// TwinCAT 3 PLC project Untitled1
// ProgramVersion: 3.1.4023.0
// libraries:
//   Tc2_MC2, * (Beckhoff Automation GmbH)
//   Tc2_NC, * (Beckhoff Automation GmbH)
//   Tc2_Standard, * (Beckhoff Automation GmbH)
//   Tc2_SUPS, * (Beckhoff Automation GmbH)
//   Tc2_System, * (Beckhoff Automation GmbH)
//   Tc2_Utilities, * (Beckhoff Automation GmbH)
//   Tc3_Module, * (Beckhoff Automation GmbH)
// project tree:
//   GVLs/ GVL.TcGVL
//   / PlcTask.TcTTO
//   POUs/ Axis1_Motion.TcPOU, Axis2_Motion.TcPOU, MAIN.TcPOU
//   POUs/PersistentFunction/ FB_Dummy.TcPOU (not stored), SLOWTASK.TcPOU (not stored), UPSPersitent.TcPOU (not stored)

CONFIGURATION Untitled1
    RESOURCE PLC ON TwinCAT3
        TASK PlcTask(INTERVAL := T#10ms, PRIORITY := 20);
        PROGRAM MAIN WITH PlcTask : MAIN;
        PROGRAM Axis1_FC WITH PlcTask : Axis1_FC;
        PROGRAM INIT WITH PlcTask : INIT;
        PROGRAM Axis2_FC WITH PlcTask : Axis2_FC;
    END_RESOURCE
END_CONFIGURATION

// ---- GVLs/GVL.TcGVL

VAR_GLOBAL
	//global   
	simulation:BOOL:=TRUE;
	btn_LocalOrRemote:BOOL:=FALSE;
	E_STOP  :BOOL;(*急停NC*) 
	E_STOP_In  AT%I*:BOOL;(*急停NC*) 
	E_STOP_rem:BOOL:=TRUE;//远程急停
	initStatus: BOOL;
	
	E_STOP_led :BOOL;(*急停指示*)
	Local_led  :BOOL;(*本地模式指示*)
	Remote_led :BOOL;(*远程模式指示*)
	Error:BOOL;
	ErrorId:INT;
	ErrorDescription:STRING;

	m_restartTC: BOOL;
	E_STOP_ftring:F_TRIG;
    E_STOP_rem_ftring:F_TRIG;
	
	//axis1
	axis1:AXIS_REF;
	LVDT1_IN AT%I*:INT;(*1#LVDT*)
	foreward_limit_axis1:BOOL;
	foreward_limit_axis1_In AT%I*:BOOL;//1#电机正向限位
	foreward_limit_axis1_simu:BOOL;//1#电机正向限位
	backward_limit_axis1 AT%I*:BOOL:=TRUE;//1#电机负向限位（准直器未加，默认为TRUE）
	touchLimitSwitch_axis1:BOOL;
	Axis1_error :BOOL;(*电机1故障指示*)
	Axis1_moving:BOOL;(*1#电机运行指示*)
	LVDT1_FunctionOn:BOOL;
	LVDT1_PV  :REAL;(*1#LVDT*)
	LVDT1_Threshold :REAL;
	LVDT1_OutOfThresholdRange :BOOL:=TRUE;
	LVDT1_OnceInRangeFlag :INT;
	LVDT1_ManualReleaseAlarm :BOOL;
	Axis1_Currentvelocity:REAL;
	btn_Move_Axis1: BOOL;
	btn_JogForward_Axis1: BOOL;
	btn_JogBackward_Axis1: BOOL;
	btn_Stop_Axis1: BOOL;
	btn_Reset_Axis1: BOOL;
	btn_SetPosition_Axis1:BOOL;
	Moving_done_Axis1:BOOL;
	PositionSetValue_Axis1:REAL;
	PositionSetDone_Axis1:BOOL;
	
	//axis2
	axis2:AXIS_REF;
	LVDT2_IN AT%I*:INT;(*2#LVDT*)
	foreward_limit_axis2:BOOL;
	foreward_limit_axis2_In AT%I*:BOOL;//2#电机正向限位
	foreward_limit_axis2_simu:BOOL;//1#电机正向限位
	backward_limit_axis2 AT%I*:BOOL:=TRUE;//2#电机负向限位（准直器未加，默认为TRUE）
	touchLimitSwitch_axis2:BOOL;
	Axis2_error :BOOL;(*电机2故障指示*)	 
	Axis2_moving	:BOOL;(*2#电机运行指示*)
	LVDT2_FunctionOn:	BOOL;	
	LVDT2_PV	:REAL;(*2#LVDT*)	
	LVDT2_Threshold	:REAL;	
	LVDT2_OutOfThresholdRange	:BOOL:=TRUE;	
	LVDT2_OnceInRangeFlag	:INT;	
	LVDT2_ManualReleaseAlarm	:BOOL;
	Axis2_Currentvelocity	:REAL;
	btn_Move_Axis2: BOOL;
	btn_JogForward_Axis2: BOOL;
	btn_JogBackward_Axis2: BOOL;
	btn_Stop_Axis2: BOOL;
	btn_Reset_Axis2: BOOL;
	btn_SetPosition_Axis2:BOOL;
	Moving_done_Axis2:BOOL;
	PositionSetValue_Axis2:REAL;
	PositionSetDone_Axis2:BOOL;
	
	//axis all
	btn_Move_AxisAll:BOOL;
	RTrig_Move_AxisAll:R_Trig;
	btn_Stop_AxisAll:BOOL;
	RTrig_Stop_AxisAll:R_Trig;
	btn_JogForward_AxisAll:BOOL;
	RTrig_JogForward_AxisAll:R_Trig;
	btn_JogBackward_AxisAll:BOOL;
	RTrig_JogBackward_AxisAll:R_Trig;
	btn_Reset_AxisAll:BOOL;
	RTrig_Reset_AxisAll:R_Trig;
 
	///
	///EPICS->PLC,Command
	///
	(*BOOL类型，占一个寄存器，存储16bit *)
	//1.global
	MOD_btn_LocalOrRemote						AT%MX0.0:BOOL;//12288.0  
	MOD_btn_E_STOP								AT%MX0.1:BOOL:=TRUE;//12288.1 
	MOD_m_restartTC								AT%MX0.2:BOOL;//12288.2 
	//2.axis1
	MOD_btn_Move_Axis1                          AT%MX2.0:BOOL;//12289.0
	MOD_btn_JogForward_Axis1                    AT%MX2.1:BOOL;//12289.1
	MOD_btn_JogBackward_Axis1                   AT%MX2.2:BOOL;//12289.2
	MOD_btn_Stop_Axis1                          AT%MX2.3:BOOL;//12289.3
	MOD_btn_Reset_Axis1                         AT%MX2.4:BOOL;//12289.4
	MOD_btn_SetPosition_Axis1                   AT%MX2.5:BOOL;//12289.5
	MOD_LVDT1_FunctionOn                        AT%MX2.6:BOOL;//12289.6
	MOD_LVDT1_ManualReleaseAlarm                AT%MX2.7:BOOL;//12289.7  
	MOD_btn_backup3       		                AT%MX3.0:BOOL;//12289.8
	MOD_btn_backup4			                    AT%MX3.1:BOOL;//12289.9
	MOD_btn_backup5                  			AT%MX3.2:BOOL;//12289.10
	MOD_btn_backup6                  			AT%MX3.3:BOOL;//12289.11
	MOD_btn_backup7                				AT%MX3.4:BOOL;//12289.12
	MOD_btn_backup8                         	AT%MX3.5:BOOL;//12289.13
	MOD_btn_backup9                				AT%MX3.6:BOOL;//12289.14
	MOD_btn_backup10	                        AT%MX3.7:BOOL;//12289.15
	(*REAL类型，每个值占两个寄存器*)   
	MOB_targetPositionAxis1                     AT%MB500:REAL;//12538
	MOB_targetVelocityAxis1                     AT%MB504:REAL;//12540
	MOB_increaseJogPositionAxis1                AT%MB508:REAL;//12542
	MOB_Axis1_minPosition                       AT%MB512:REAL;//12544
	MOB_Axis1_maxPosition                       AT%MB516:REAL;//12546
	MOD_LVDT1_Threshold                         AT%MB520:REAL;//12548
	MOD_PositionSetValue_Axis1					AT%MB524:REAL;//12550
	//3.axis2
	MOD_btn_Move_Axis2                          AT%MX4.0:BOOL;//12290.0
	MOD_btn_JogForward_Axis2                    AT%MX4.1:BOOL;//12290.1
	MOD_btn_JogBackward_Axis2                   AT%MX4.2:BOOL;//12290.2
	MOD_btn_Stop_Axis2                          AT%MX4.3:BOOL;//12290.3
	MOD_btn_Reset_Axis2                         AT%MX4.4:BOOL;//12290.4
	MOD_btn_SetPosition_Axis2                   AT%MX4.5:BOOL;//12290.5
	MOD_LVDT2_FunctionOn			            AT%MX4.6:BOOL;//12290.6
	MOD_LVDT2_ManualReleaseAlarm                AT%MX4.7:BOOL;//12290.7  
	MOD_btn_backup13       		                AT%MX5.0:BOOL;//12290.8
	MOD_btn_backup14			                AT%MX5.1:BOOL;//12290.9
	MOD_btn_backup15                  			AT%MX5.2:BOOL;//12290.10
	MOD_btn_backup16                  			AT%MX5.3:BOOL;//12290.11
	MOD_btn_backup17                			AT%MX5.4:BOOL;//12290.12
	MOD_btn_backup18                         	AT%MX5.5:BOOL;//12290.13
	MOD_btn_backup19                			AT%MX5.6:BOOL;//12290.14
	MOD_btn_backup20	                        AT%MX5.7:BOOL;//12290.15
	(*REAL类型，每个值占两个寄存器*)   
	MOB_targetPositionAxis2                     AT%MB600:REAL;//12588
	MOB_targetVelocityAxis2                     AT%MB604:REAL;//12590
	MOB_increaseJogPositionAxis2                AT%MB608:REAL;//12592
	MOB_Axis2_minPosition                       AT%MB612:REAL;//12594
	MOB_Axis2_maxPosition                       AT%MB616:REAL;//12596
	MOD_LVDT2_Threshold                         AT%MB620:REAL;//12598
	MOD_PositionSetValue_Axis2					AT%MB624:REAL;//12600
	//4. aixs all
	MOD_btn_Move_AxisAll                        AT%MX6.0:BOOL;//12291.0
	MOD_btn_JogForward_AxisAll                  AT%MX6.1:BOOL;//12291.1
	MOD_btn_JogBackward_AxisAll                 AT%MX6.2:BOOL;//12291.2
	MOD_btn_Stop_AxisAll                        AT%MX6.3:BOOL;//12291.3
	MOD_btn_Reset_AxisAll                       AT%MX6.4:BOOL;//12291.3
	///
	///PLC->EPICS,Response
	///
	//1.global
	(*BOOL类型，占一个寄存器，存储16bit*)
	MOD_E_STOP_led                              AT%MX10.0:BOOL;//12293.0  
	MOD_Local_led                               AT%MX10.1:BOOL;//12293.1 
	MOD_Remote_led                              AT%MX10.2:BOOL;//12293.2 
	MOD_Error_led								AT%MX10.3:BOOL;//12293.3 
	//2.axis1
	MOD_Axis1_error                             AT%MX12.0:BOOL;//12294.0
	MOD_Axis1_moving                            AT%MX12.1:BOOL;//12294.1
	MOD_foreward_limit_axis1                   	AT%MX12.2:BOOL;//12294.2
	MOD_backward_limit_axis1                    AT%MX12.3:BOOL;//12294.3
	MOD_Moving_done_Axis1                       AT%MX12.4:BOOL;//12294.4
	MOD_PositionSetDone_Axis1	                AT%MX12.5:BOOL;//12294.5
	MOD_B_Backup2	   			                AT%MX12.6:BOOL;//12294.6	
	MOD_B_Backup3	   			                AT%MX12.7:BOOL;//12294.7 
	MOD_B_Backup4                             	AT%MX13.0:BOOL;//12294.8
	MOD_B_Backup5                            	AT%MX13.1:BOOL;//12294.9
	MOD_B_Backup6                   			AT%MX13.2:BOOL;//12294.10
	MOD_B_Backup7                    			AT%MX13.3:BOOL;//12294.11
	MOD_B_Backup8                      			AT%MX13.4:BOOL;//12294.12
	MOD_B_Backup9	   			                AT%MX13.5:BOOL;//12294.13	
	MOD_B_Backup10	   			                AT%MX13.6:BOOL;//12294.14 	
	MOD_B_Backup11	   			                AT%MX13.7:BOOL;//12294.15	
	(*REAL类型，每个值占两个寄存器*) 
	MOD_Axis1_Currentvelocity                   AT%MB700:REAL;//12638
	MOD_Axis1_CurrentPosition                   AT%MB704:REAL;//12640
 	MOD_LVDT1_PV 	                            AT%MB708:REAL;//12642
	//3.axis2
	MOD_Axis2_error                             AT%MX14.0:BOOL;//12295.0
	MOD_Axis2_moving                            AT%MX14.1:BOOL;//12295.1
	MOD_foreward_limit_axis2                   	AT%MX14.2:BOOL;//12295.2
	MOD_backward_limit_axis2                    AT%MX14.3:BOOL;//12295.3
	MOD_Moving_done_Axis2                       AT%MX14.4:BOOL;//12295.4
	MOD_PositionSetDone_Axis2	                AT%MX14.5:BOOL;//12295.5
	MOD_B_Backup13	   			                AT%MX14.6:BOOL;//12295.6 	
	MOD_B_Backup14	   			                AT%MX14.7:BOOL;//12295.7	 
	MOD_B_Backup15                            	AT%MX15.0:BOOL;//12295.8
	MOD_B_Backup16                            	AT%MX15.1:BOOL;//12295.9
	MOD_B_Backup17                   			AT%MX15.2:BOOL;//12295.10
	MOD_B_Backup18                    			AT%MX15.3:BOOL;//12295.11
	MOD_B_Backup19                      		AT%MX15.4:BOOL;//12295.12
	MOD_B_Backup20	   			                AT%MX15.5:BOOL;//12295.13
	MOD_B_Backup21	   			                AT%MX15.6:BOOL;//12295.14
	MOD_B_Backup22	   			                AT%MX15.7:BOOL;//12295.15
	// REAL类型，每个值占两个寄存器  
	// REAL类型，每个值占两个寄存器  
	MOD_Axis2_Currentvelocity                	AT%MB800:REAL;//12688
	MOD_Axis2_CurrentPosition                   AT%MB804:REAL;//12690
 	MOD_LVDT2_PV                                AT%MB808:REAL;//12692
	// REAL类型，每个值占两个寄存器  
	MOD_ErrorId				                	AT%MB812:REAL;//12694
END_VAR

VAR_GLOBAL PERSISTENT
	//Axis1
    Axis1_CurrentPosition_retain:REAL;
	Axis1_minPosition		:REAL;
	Axis1_maxPosition		:REAL;
    increaseJogPositionAxis1:REAL;
	targetVelocityAxis1: REAL;
	targetPositionAxis1: REAL;
	//axis2
	Axis2_CurrentPosition_retain:REAL;
	Axis2_minPosition		:REAL;   
	Axis2_maxPosition		:REAL;
	increaseJogPositionAxis2:REAL;
	targetVelocityAxis2: REAL;
	targetPositionAxis2: REAL;
END_VAR

// ---- POUs/MAIN.TcPOU
PROGRAM MAIN
VAR
	//
	//Gloabal
	//
	RestartTC: TC_Restart;
	//
	//init
	//
	SetPosition_delay     	  :TON;
	SetPosition2getCurrentPositiondelay     	  :TON;
	init_State: INT;
	MC_SetPosition_Axis1: MC_SetPosition;
	MC_SetPosition_Axis2: MC_SetPosition;

	m_State_AxisAll: INT;
	m_delay:TON;
	init_dalay:TON;
END_VAR

//初始化，存储位置写入当前位置灯
A_init();
IF initStatus THEN
	//Axis1运动
	Axis1_Motion();
	//Axis2运动
	Axis2_Motion();
	//All Axis运动
	AxisAll_Motion();
END_IF
//是否simulation
simu();
//数据persistent存储
UPSPersitent();
//RestartTC
A_RestartTC();
//LVDT
LVDT();
//modbus
modbus();
//
limitSwicth();

ACTION A_init:
//
//0.delay
//
//
init_dalay.PT:=T#3S;
init_dalay();
init_dalay.IN:=TRUE;
IF NOT init_dalay.Q THEN
	RETURN;
END_IF
//1.初始化：加载保存的persistent变量：位置，并写入当前位置
//
init_MC();
SetPosition_delay.PT:=T#1S;
SetPosition_delay();
CASE init_State OF 
	0:
		IF NOT Axis1_moving AND NOT  Axis2_moving THEN
			init_State:=1;
		END_IF
	1:
		IF NOT initStatus THEN
			MC_SetPosition_Axis1.Position:=Axis1_CurrentPosition_retain;
			MC_SetPosition_Axis2.Position:=	Axis2_CurrentPosition_retain;
			MC_SetPosition_Axis1.Execute:=TRUE;
			MC_SetPosition_Axis2.Execute:=TRUE;
			SetPosition_delay.IN:=TRUE;
			init_State:=2;
		END_IF
	2:
		IF MC_SetPosition_Axis1.Done AND MC_SetPosition_Axis2.Done THEN
			init_State:=88;
		END_IF
		IF SetPosition_delay.Q THEN//延时结束时，还没有设置位置成功
			init_State:=-100;
		END_IF
	88:
		initStatus:=TRUE;
		MC_SetPosition_Axis1.Execute:=FALSE;
		MC_SetPosition_Axis2.Execute:=FALSE;
		SetPosition_delay.IN:=FALSE;
		init_State:=0;
	-100:
		initStatus:=FALSE;
		SetPosition_delay.IN:=FALSE;
		MC_SetPosition_Axis1.Execute:=FALSE;
		MC_SetPosition_Axis2.Execute:=FALSE;
		Error:=TRUE;
		ErrorId:=1;
		ErrorDescription:='init fail';
END_CASE

//
//2.位置写入后，当前位置和速度即从轴中获取
//
IF initStatus THEN
	Axis1_CurrentPosition_retain  :=LREAL_TO_REAL(axis1.NcToPlc.ActPos);
	Axis1_Currentvelocity  :=LREAL_TO_REAL(axis1.NcToPlc.ActVelo);
	Axis2_CurrentPosition_retain  :=LREAL_TO_REAL(axis2.NcToPlc.ActPos);
	Axis2_Currentvelocity  :=LREAL_TO_REAL(axis2.NcToPlc.ActVelo);
END_IF
END_ACTION

ACTION A_RestartTC:
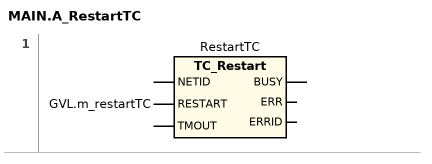
// NETWORK 1
RestartTC(RESTART := GVL.m_restartTC); // TC_Restart
END_ACTION

ACTION AxisAll_Motion:
RTrig_Move_AxisAll(CLK:=btn_Move_AxisAll,Q=>);
IF RTrig_Move_AxisAll.Q THEN
	btn_Move_Axis1:=TRUE;
	btn_Move_Axis2:=TRUE;
END_IF

RTrig_Stop_AxisAll(CLK:=btn_Stop_AxisAll,Q=>);
IF RTrig_Stop_AxisAll.Q THEN
	btn_Stop_Axis1:=TRUE;
	btn_Stop_Axis2:=TRUE;
END_IF
RTrig_JogForward_AxisAll(CLK:=btn_JogForward_AxisAll,Q=>);
IF RTrig_JogForward_AxisAll.Q THEN
	btn_JogForward_Axis1:=TRUE;
	btn_JogForward_Axis2:=TRUE;
END_IF
RTrig_JogBackward_AxisAll(CLK:=btn_JogBackward_AxisAll,Q=>);
IF RTrig_JogBackward_AxisAll.Q THEN
	btn_JogBackward_Axis1:=TRUE;
	btn_JogBackward_Axis2:=TRUE;
END_IF
RTrig_Reset_AxisAll(CLK:=btn_Reset_AxisAll,Q=>);
IF RTrig_Reset_AxisAll.Q THEN
	btn_Reset_Axis1:=TRUE;
	btn_Reset_Axis2:=TRUE;
END_IF
END_ACTION

ACTION init_MC:
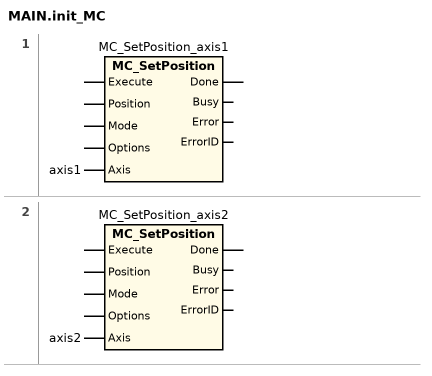
// NETWORK 1
MC_SetPosition_axis1(Axis := axis1); // MC_SetPosition

// NETWORK 2
MC_SetPosition_axis2(Axis := axis2); // MC_SetPosition
END_ACTION

ACTION limitSwicth:
touchLimitSwitch_axis1:=foreward_limit_axis1 AND backward_limit_axis1;
touchLimitSwitch_axis2:=foreward_limit_axis2 AND backward_limit_axis2;
END_ACTION

ACTION LVDT:
LVDT1_PV:=INT_TO_REAL(LVDT1_IN);
LVDT2_PV:=INT_TO_REAL(LVDT2_IN);
//LVDT1
IF LVDT1_FunctionOn THEN
	IF LVDT1_PV<=LVDT1_Threshold THEN//进入传感器限位区，报错
		LVDT1_OutOfThresholdRange:=FALSE;
		Error:=TRUE;
		ErrorDescription:='LVDT1 In Alarm Range';
		LVDT1_OnceInRangeFlag:=1;//标志曾经进入过限位区
	END_IF
	//正常情况下，出限位区，恢复正常
	//如果曾经进入过限位区，需要手动解除后，报警才解除
	IF LVDT1_OnceInRangeFlag=1 THEN
		LVDT1_OutOfThresholdRange:=FALSE;
		Error:=TRUE;
		ErrorDescription:='LVDT1 In Alarm Range';
		IF LVDT1_ManualReleaseAlarm THEN
			Error:=FALSE;
			ErrorDescription:='';
			LVDT1_OnceInRangeFlag:=0;
			LVDT1_ManualReleaseAlarm:=FALSE;
			LVDT1_OutOfThresholdRange:=TRUE;
		END_IF
	END_IF
END_IF
//LVDT2
IF LVDT2_FunctionOn THEN
	IF LVDT2_PV<=LVDT2_Threshold THEN//进入传感器限位区，报错
		LVDT2_OutOfThresholdRange:=FALSE;
		Error:=TRUE;
		ErrorDescription:='LVDT2 In Alarm Range';
		LVDT2_OnceInRangeFlag:=1;//标志曾经进入过限位区
	END_IF
	//正常情况下，出限位区，恢复正常
	//如果曾经进入过限位区，需要手动解除后，报警才解除
	IF LVDT2_OnceInRangeFlag=1 THEN
		LVDT2_OutOfThresholdRange:=FALSE;
		Error:=TRUE;
		ErrorDescription:='LVDT2 In Alarm Range';
		IF LVDT2_ManualReleaseAlarm THEN
			Error:=FALSE;
			ErrorDescription:='';
			LVDT2_OnceInRangeFlag:=0;
			LVDT2_ManualReleaseAlarm:=FALSE;
			LVDT2_OutOfThresholdRange:=TRUE;
		END_IF
	END_IF
END_IF
END_ACTION

ACTION modbus:
//PLC->EPICS，持续通讯
MOD_E_STOP_led            			:=E_STOP_led;
MOD_Axis1_error            			:=Axis1_error;
MOD_Axis2_error            			:=Axis2_error;
MOD_Axis1_moving           			:=Axis1_moving;
MOD_Axis2_moving           			:=Axis2_moving;
MOD_Moving_done_Axis1      			:=Moving_done_Axis1;
MOD_Moving_done_Axis2     			:=Moving_done_Axis2;
MOD_foreward_limit_axis1   			:=foreward_limit_axis1;
MOD_backward_limit_axis1   			:=backward_limit_axis1;
MOD_foreward_limit_axis2   			:=foreward_limit_axis2;
MOD_backward_limit_axis2   			:=backward_limit_axis2;
MOD_Axis1_Currentvelocity  			:=Axis1_Currentvelocity;
MOD_Axis2_Currentvelocity  			:=Axis2_Currentvelocity;
MOD_Axis1_CurrentPosition  			:=Axis1_CurrentPosition_retain;
MOD_Axis2_CurrentPosition  			:=Axis2_CurrentPosition_retain;
MOD_LVDT1_PV               			:=LVDT1_PV;
MOD_LVDT2_PV               			:=LVDT2_PV;
MOD_PositionSetDone_Axis1			:=PositionSetDone_Axis1;
MOD_PositionSetDone_Axis2			:=PositionSetDone_Axis2;
MOD_Error_led						:=Error;
MOD_ErrorId							:=ErrorId;
//EPICS->PLC，持续通讯
//btn_LocalOrRemote					:=MOD_btn_LocalOrRemote;

//本地模式切换
IF btn_LocalOrRemote THEN
	Local_led:= TRUE;
	Remote_led:=FALSE;
ELSE	
	Local_led:= FALSE;
	Remote_led:=TRUE;
END_IF;
MOD_Local_led:=Local_led;
MOD_Remote_led:=Remote_led;
//远程开关开，通讯
IF  MOD_Remote_led  THEN   
	//global 
	m_restartTC						:=MOD_m_restartTC;
	E_STOP_rem						:=MOD_btn_E_STOP;
	//axis1
	LVDT1_FunctionOn             	:=MOD_LVDT1_FunctionOn;    
	LVDT1_ManualReleaseAlarm     	:=MOD_LVDT1_ManualReleaseAlarm; 
	btn_SetPosition_Axis1           :=MOD_btn_SetPosition_Axis1;
	targetPositionAxis1				:=MOB_targetPositionAxis1;
	targetVelocityAxis1				:=MOB_targetVelocityAxis1;
	increaseJogPositionAxis1		:=MOB_increaseJogPositionAxis1;
	Axis1_minPosition				:=MOB_Axis1_minPosition;
	Axis1_maxPosition				:=MOB_Axis1_maxPosition;
	LVDT1_Threshold             	:=MOD_LVDT1_Threshold;
	PositionSetValue_Axis1			:=MOD_PositionSetValue_Axis1;
	//axis2
	LVDT2_Threshold              	:=MOD_LVDT2_Threshold;
	LVDT2_FunctionOn             	:=MOD_LVDT2_FunctionOn;    
	LVDT2_ManualReleaseAlarm    	:=MOD_LVDT2_ManualReleaseAlarm; 
	btn_SetPosition_Axis2           :=MOD_btn_SetPosition_Axis2;
	targetPositionAxis2				:=MOB_targetPositionAxis2;
	targetVelocityAxis2				:=MOB_targetVelocityAxis2;
	increaseJogPositionAxis2		:=MOB_increaseJogPositionAxis2;
	Axis2_minPosition				:=MOB_Axis2_minPosition;
	Axis2_maxPosition				:=MOB_Axis2_maxPosition;
	LVDT2_Threshold             	:=MOD_LVDT2_Threshold;
	PositionSetValue_Axis2			:=MOD_PositionSetValue_Axis2;
	//axis all
	btn_Move_AxisAll				:=MOD_btn_Move_AxisAll;
	btn_JogForward_AxisAll			:=MOD_btn_JogForward_AxisAll;
	btn_JogBackward_AxisAll			:=MOD_btn_JogBackward_AxisAll;
	btn_Stop_AxisAll				:=MOD_btn_Stop_AxisAll;
	IF NOT MOD_btn_Move_AxisAll	THEN
			btn_Move_Axis1                	:=MOD_btn_Move_Axis1;
			btn_Move_Axis2                	:=MOD_btn_Move_Axis2;
	ELSE
		btn_Move_AxisAll:=TRUE;
	END_IF
		IF NOT MOD_btn_Stop_AxisAll	THEN
			btn_Stop_Axis1                	:=MOD_btn_Stop_Axis1;
			btn_Stop_Axis2                	:=MOD_btn_Stop_Axis2;
	ELSE
		btn_Stop_AxisAll:=TRUE;
	END_IF
	IF NOT MOD_btn_JogForward_AxisAll	THEN
			btn_JogForward_Axis1              :=MOD_btn_JogForward_Axis1;
			btn_JogForward_Axis2              :=MOD_btn_JogForward_Axis2;
	ELSE
		btn_JogForward_AxisAll:=TRUE;
	END_IF
	IF NOT MOD_btn_JogBackward_AxisAll	THEN
			btn_JogBackward_Axis1                	:=MOD_btn_JogBackward_Axis1;
			btn_JogBackward_Axis2                	:=MOD_btn_JogBackward_Axis2;
	ELSE
		btn_JogBackward_AxisAll:=TRUE;
	END_IF
	IF NOT MOD_btn_Reset_AxisAll	THEN
			btn_Reset_Axis1                	:=MOD_btn_Reset_Axis1;
			btn_Reset_Axis2                	:=MOD_btn_Reset_Axis2;
	ELSE
		btn_Reset_AxisAll:=TRUE;
	END_IF
ELSE
	MOB_Axis1_minPosition				:=Axis1_minPosition;
	MOB_Axis1_maxPosition				:=Axis1_maxPosition;
	MOB_Axis2_minPosition				:=Axis2_minPosition;
	MOB_Axis2_maxPosition				:=Axis2_maxPosition;
	MOB_targetPositionAxis1				:=targetPositionAxis1;
	MOB_targetVelocityAxis1				:=targetVelocityAxis1;
	MOB_increaseJogPositionAxis1		:=increaseJogPositionAxis1;
	MOB_targetPositionAxis2				:=targetPositionAxis2;
	MOB_targetVelocityAxis2				:=targetVelocityAxis2;
	MOB_increaseJogPositionAxis2		:=increaseJogPositionAxis2;
END_IF
END_ACTION

ACTION simu:
IF simulation THEN
	E_STOP:=TRUE;
	foreward_limit_axis1:=TRUE;
	foreward_limit_axis2:=TRUE;
ELSE
	E_STOP:=E_STOP_In;
	foreward_limit_axis1:=foreward_limit_axis1_In;
	foreward_limit_axis2:=foreward_limit_axis2_In;
END_IF
END_ACTION

END_PROGRAM

// ---- POUs/Axis1_Motion.TcPOU
PROGRAM Axis1_Motion
VAR
	//power
	MC_Power_Axis1: MC_Power;
	//Move
	m_State_Axis1: INT;
	MC_MoveAbsolute_Axis1: MC_MoveAbsolute;

	//JOG
	j_State_Axis1: INT;
	MC_JOG_Axis1: MC_Jog;

	//Stop
	MC_Stop_Axis1: MC_Stop;
	s_State_Axis1: INT;

	//reset
	r_State_Axis1: INT;
	MC_Reset_Axis1: MC_Reset;

	//setposition
	MC_SetPosition_Axis1: MC_SetPosition;
	sp_State_Axis1: INT;
	SetPosition_delay_Axis1:TON;

	//button interlock
	Axis1_J1: BOOL;//JOG+
	Axis1_J2: BOOL;//JOG-
	Axis1_P: BOOL;//Position moving
	Axis1_S: BOOL;//Stop
	Axis1_SP: BOOL;//set position
	//input protect
	Axis1_PositionProtectionSet:BOOL;
	Axis1_InputPositionOutOfRange:BOOL;
END_VAR

//
//输入保护
//
IF targetPositionAxis1>=Axis1_minPosition AND targetPositionAxis1<=Axis1_maxPosition THEN
	Axis1_InputPositionOutOfRange:=FALSE;
	Error:=FALSE;
	ErrorId:=0;
	ErrorDescription:='';
ELSE
	Axis1_InputPositionOutOfRange:=TRUE;
	Error:=TRUE;
	ErrorId:=1001;
	ErrorDescription:='Axis1_InputPositionOutOfRange';
	RETURN;
END_IF
//
//运行状态指示
//
Axis1.ReadStatus();
IF  Axis1.Status.Moving  THEN
	Axis1_moving:=TRUE;
ELSE
	Axis1_moving:=FALSE;
END_IF;
//
//电机错误指示
//
IF  axis1.NcToPlc.ErrorCode=0 THEN
	Axis1_error     := FALSE;
ELSE
	Axis1_error     := TRUE;
	Error:=TRUE;
	ErrorId:=1002;
	ErrorDescription:='axis1.NcToPlc.ErrorCode=0';
END_IF;
//
//Moving_done_Axis1
//
//
Moving_done_Axis1:=MC_MoveAbsolute_Axis1.Done OR MC_JOG_Axis1.Done;

//Positioning move
//
A_MCAxis1();
CASE m_State_Axis1 OF 
	0:
		//检查是否有错误等
		IF  E_STOP  AND NOT Axis1_error THEN
			m_State_Axis1:=1;
		ELSE
			m_State_Axis1:=-100;
		END_IF
	1:
		//检查电机是否已经上电，如无，则上电
		IF 	NOT MC_Power_Axis1.Status THEN
			MC_Power_Axis1.Enable:=TRUE;
		ELSE
			m_State_Axis1:=2;
		END_IF
	2:
		//定位运行
		MC_MoveAbsolute_Axis1.Position:=targetPositionAxis1;
		MC_MoveAbsolute_Axis1.Velocity:=targetVelocityAxis1;
		IF btn_Move_Axis1 THEN
			MC_MoveAbsolute_Axis1.Execute:=TRUE;
			m_State_Axis1:=3;
		END_IF
	3:
		//是否运动到位
		IF MC_MoveAbsolute_Axis1.Done THEN
			m_State_Axis1:=88;
		END_IF
	88:
		btn_Move_Axis1:=FALSE;
		MC_MoveAbsolute_Axis1.Execute:=FALSE;
		m_State_Axis1:=0;		
	-100:
		btn_Move_Axis1:=FALSE;
		MC_MoveAbsolute_Axis1.Execute:=FALSE;
		Error:=TRUE;
		ErrorId:=1002;
		ErrorDescription:='E_STOP AND NOT Axis1_error';
		
END_CASE
//
//JOG+
//
CASE j_State_Axis1 OF 
	0:
		//检查是否有错误等
		IF  E_STOP  AND NOT Axis1_error THEN
			j_State_Axis1:=1;
		ELSE
			j_State_Axis1:=-100;
		END_IF
	1:
		//检查电机是否已经上电，如无，则上电
		IF 	NOT MC_Power_Axis1.Status THEN
			MC_Power_Axis1.Enable:=TRUE;
		ELSE
			j_State_Axis1:=2;
		END_IF
	2:
		//JOG运行
		MC_JOG_Axis1.Position:=increaseJogPositionAxis1;
		MC_JOG_Axis1.Velocity:=targetVelocityAxis1;
		IF btn_JogForward_Axis1 AND NOT btn_JogBackward_Axis1 THEN
			MC_JOG_Axis1.JogForward:=TRUE;
			j_State_Axis1:=3;
		END_IF
		IF btn_JogBackward_Axis1 AND NOT btn_JogForward_Axis1 THEN
			MC_JOG_Axis1.JogBackwards:=TRUE;
			j_State_Axis1:=3;
		END_IF
	3:
		//是否运动到位
		IF btn_JogForward_Axis1 THEN
			btn_JogForward_Axis1:=FALSE;
		END_IF 
		IF btn_JogBackward_Axis1 THEN
			btn_JogBackward_Axis1:=FALSE;
		END_IF
		IF MC_JOG_Axis1.Done THEN
			j_State_Axis1:=88;
		END_IF
	88:
		MC_JOG_Axis1.JogForward:=FALSE;
		MC_JOG_Axis1.JogBackwards:=FALSE;
		btn_JogForward_Axis1:=FALSE;
		btn_JogBackward_Axis1:=FALSE;
		j_State_Axis1:=0;	
		
	-100:
		MC_JOG_Axis1.JogForward:=FALSE;
		MC_JOG_Axis1.JogBackwards:=FALSE;
		btn_JogForward_Axis1:=FALSE;
		btn_JogBackward_Axis1:=FALSE;
		Error:=TRUE;
		ErrorId:=1002;
		ErrorDescription:='E_STOP AND NOT Axis1_error';	
END_CASE
//
//STOP
//
CASE s_State_Axis1 OF 
	0:
		//检查是否有错误等
		IF  E_STOP  AND NOT Axis1_error THEN
			s_State_Axis1:=1;
		ELSE
			s_State_Axis1:=-100;
		END_IF
	1:
		//检查电机是否已经上电，如无，则上电
		IF 	NOT MC_Power_Axis1.Status THEN
			MC_Power_Axis1.Enable:=TRUE;
		ELSE
			s_State_Axis1:=2;
		END_IF
	2:
		//STOP
		IF btn_Stop_Axis1 THEN
			MC_Stop_Axis1.Execute:=TRUE;
			s_State_Axis1:=3;
		END_IF
	3:
		//是否运动到位
		IF MC_Stop_Axis1.Done THEN
			s_State_Axis1:=88;
		END_IF
	88:
		btn_Stop_Axis1:=FALSE;
		MC_Stop_Axis1.Execute:=FALSE;
		s_State_Axis1:=0;	
		//reset status
		btn_Move_Axis1:=FALSE;
		MC_MoveAbsolute_Axis1.Execute:=FALSE;
		btn_JogForward_Axis1:=FALSE;
		btn_JogBackward_Axis1:=FALSE;
		MC_JOG_Axis1.JogForward:=FALSE;
		MC_JOG_Axis1.JogBackwards:=FALSE;
		m_State_Axis1:=0;
		j_State_Axis1:=0;
	-100:
		btn_Stop_Axis1:=FALSE;
		MC_Stop_Axis1.Execute:=FALSE;
		Error:=TRUE;
		ErrorId:=1002;
		ErrorDescription:='E_STOP AND NOT Axis1_error';
		//reset status
		btn_Move_Axis1:=FALSE;
		MC_MoveAbsolute_Axis1.Execute:=FALSE;
		btn_JogForward_Axis1:=FALSE;
		btn_JogBackward_Axis1:=FALSE;
		MC_JOG_Axis1.JogForward:=FALSE;
		MC_JOG_Axis1.JogBackwards:=FALSE;
		m_State_Axis1:=0;
		j_State_Axis1:=0;
END_CASE
//
//Reset
//
CASE r_State_Axis1 OF 
	0:
		IF btn_Reset_Axis1 THEN
			MC_Reset_Axis1.Execute:=TRUE;
			r_State_Axis1:=1;
		END_IF
	1:
		//是否运动到位
		IF MC_Reset_Axis1.Done THEN
			r_State_Axis1:=88;
		END_IF
	88:
		r_State_Axis1:=0;
		MC_Reset_Axis1.Execute:=FALSE;	
		btn_Reset_Axis1:=FALSE;
		//reset status
		btn_Move_Axis1:=FALSE;
		MC_MoveAbsolute_Axis1.Execute:=FALSE;
		btn_JogForward_Axis1:=FALSE;
		btn_JogBackward_Axis1:=FALSE;
		MC_JOG_Axis1.JogForward:=FALSE;
		MC_JOG_Axis1.JogBackwards:=FALSE;
		m_State_Axis1:=0;
		s_State_Axis1:=0;
		j_State_Axis1:=0;
END_CASE
//
//setposotion
//
SetPosition_delay_Axis1.PT:=T#0.1S;
SetPosition_delay_Axis1();
IF btn_SetPosition_Axis1 THEN
	CASE sp_State_Axis1 OF 
		0:
			IF NOT Axis1_moving THEN
				sp_State_Axis1:=1;
			END_IF
		1:
			MC_SetPosition_Axis1.Position:=PositionSetValue_Axis1;
			MC_SetPosition_Axis1.Execute:=TRUE;
			SetPosition_delay_Axis1.IN:=TRUE;
			sp_State_Axis1:=2;
		2:
			IF MC_SetPosition_Axis1.Done THEN
				sp_State_Axis1:=88;
			END_IF
			IF SetPosition_delay_Axis1.Q THEN//延时结束时，还没有设置位置成功
				sp_State_Axis1:=-100;
			END_IF
		88:
			PositionSetDone_Axis1:=TRUE;
			MC_SetPosition_Axis1.Execute:=FALSE;
			SetPosition_delay_Axis1.IN:=FALSE;
			sp_State_Axis1:=0;
			btn_SetPosition_Axis1:=FALSE;
		-100:
			PositionSetDone_Axis1:=FALSE;
			MC_SetPosition_Axis1.Execute:=FALSE;
			SetPosition_delay_Axis1.IN:=FALSE;
			btn_SetPosition_Axis1:=FALSE;
	END_CASE
END_IF
//
//屏幕按钮**互锁变量,FALSE时，该按钮灰色不能触发
//
//J1->JOG+
IF  foreward_limit_axis1 AND E_STOP  AND Local_led AND NOT  Axis1_error  AND NOT  Axis1_moving AND
	NOT btn_Move_Axis1 AND NOT  btn_JogBackward_Axis1  THEN
	Axis1_J1     := TRUE;
ELSE
	Axis1_J1     := FALSE;
END_IF;
//J2>JOG-
IF  backward_limit_axis1  AND E_STOP   AND Local_led AND NOT  Axis1_error  AND NOT  Axis1_moving AND 
	 NOT  btn_Move_Axis1 AND NOT btn_JogForward_Axis1 THEN
	Axis1_J2     := TRUE;
ELSE
	Axis1_J2     := FALSE;
END_IF;
//P->PositionMove
IF  E_STOP   AND Local_led AND NOT  Axis1_error  AND NOT  Axis1_moving AND 
	 NOT btn_JogForward_Axis1  AND NOT  btn_JogBackward_Axis1 THEN
	Axis1_P     := TRUE;
ELSE
	Axis1_P     := FALSE;
END_IF;
//SP->SetPosition
IF E_STOP  AND Local_led AND NOT  Axis1_error  AND NOT Axis1_moving  THEN
	Axis1_SP     := TRUE;
ELSE
	Axis1_SP     := FALSE;
END_IF;
//S->Stop
IF E_STOP  AND Local_led AND NOT  Axis1_error THEN
	Axis1_S     := TRUE;
ELSE
	Axis1_S     := FALSE;
END_IF;
//
//
//
//急停
E_STOP_ftring(CLK:=E_STOP , Q=> );
E_STOP_rem_ftring(CLK:=E_STOP_rem , Q=> );
IF E_STOP_ftring.Q OR E_STOP_rem_ftring.Q THEN     
	E_STOP_led:= TRUE;	
	MC_Power_Axis1.Enable:=FALSE;//电机1断电
	btn_Stop_Axis1:=TRUE;//STOP axis1
	A_MCAxis1();
	Error:=TRUE;
	ErrorId:=101;
	ErrorDescription:='E_STOP';
END_IF;

ACTION A_MCAxis1:
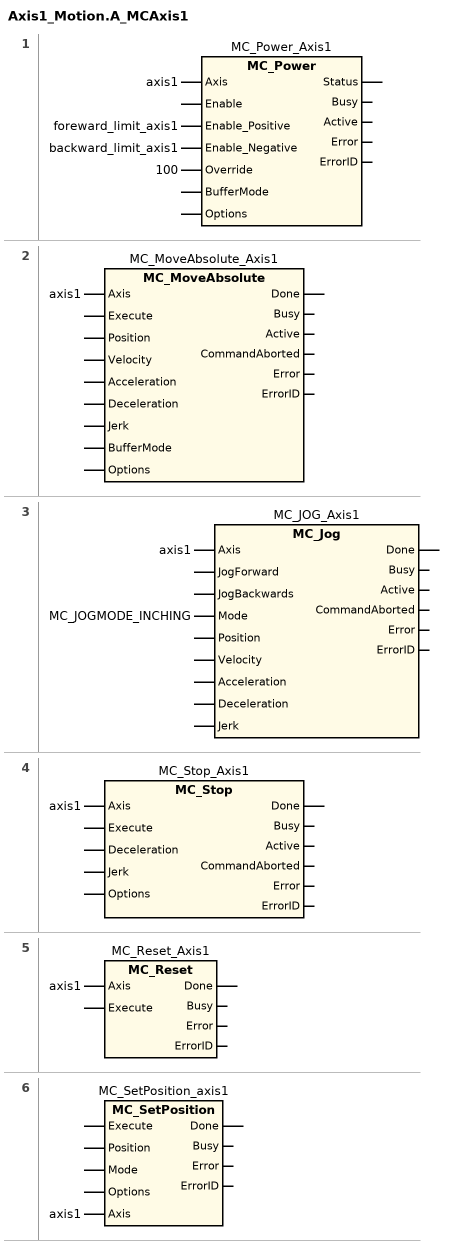
// NETWORK 1
MC_Power_Axis1(
    Axis := axis1,
    Enable_Positive := foreward_limit_axis1,
    Enable_Negative := backward_limit_axis1,
    Override := 100); // MC_Power

// NETWORK 2
MC_MoveAbsolute_Axis1(Axis := axis1); // MC_MoveAbsolute

// NETWORK 3
MC_JOG_Axis1(Axis := axis1, Mode := MC_JOGMODE_INCHING); // MC_Jog

// NETWORK 4
MC_Stop_Axis1(Axis := axis1); // MC_Stop

// NETWORK 5
MC_Reset_Axis1(Axis := axis1); // MC_Reset

// NETWORK 6
MC_SetPosition_axis1(Axis := axis1); // MC_SetPosition
END_ACTION

END_PROGRAM

// ---- POUs/Axis2_Motion.TcPOU
PROGRAM Axis2_Motion
VAR
	//power
	MC_Power_Axis2: MC_Power;
	//Move
	m_State_Axis2: INT;
	MC_MoveAbsolute_Axis2: MC_MoveAbsolute;

	//JOG
	j_State_Axis2: INT;
	MC_JOG_Axis2: MC_Jog;

	//Stop
	MC_Stop_Axis2: MC_Stop;
	s_State_Axis2: INT;

	//reset
	r_State_Axis2: INT;
	MC_Reset_Axis2: MC_Reset;

	//setposition
	MC_SetPosition_Axis2: MC_SetPosition;
	sp_State_Axis2: INT;
	SetPosition_delay_Axis2:TON;
	//button interlock
	Axis2_J1: BOOL;//JOG+
	Axis2_J2: BOOL;//JOG-
	Axis2_P: BOOL;//Position moving
	Axis2_S: BOOL;//Stop
	Axis2_SP: BOOL;//set position
	//input protect
	Axis2_PositionProtectionSet:BOOL;
	Axis2_InputPositionOutOfRange:BOOL;	
	//
END_VAR

//
//输入保护
//
IF targetPositionAxis2>=Axis2_minPosition AND targetPositionAxis2<=Axis2_maxPosition THEN
	Axis2_InputPositionOutOfRange:=FALSE;
	Error:=FALSE;
	ErrorId:=0;
	ErrorDescription:='';
ELSE
	Axis2_InputPositionOutOfRange:=TRUE;
	Error:=TRUE;
	ErrorId:=1001;
	ErrorDescription:='Axis2_InputPositionOutOfRange';
	RETURN;
END_IF
//
//运行状态指示
//
Axis2.ReadStatus();
IF  Axis2.Status.Moving  THEN
	Axis2_moving:=TRUE;
ELSE
	Axis2_moving:=FALSE;
END_IF;
//
//电机错误指示
//
IF  axis2.NcToPlc.ErrorCode=0 THEN
	Axis2_error     := FALSE;
ELSE
	Axis2_error     := TRUE;
	Error:=TRUE;
	ErrorId:=1002;
	ErrorDescription:='axis1.NcToPlc.ErrorCode=0';
END_IF;
//
//Moving_done_Axis2
//
//
Moving_done_Axis2:=MC_MoveAbsolute_Axis2.Done OR MC_JOG_Axis2.Done;
//
//Positioning move
//
A_MCAxis2();
CASE m_State_Axis2 OF 
	0:
		//检查是否有错误等
		IF  E_STOP  AND NOT Axis2_error THEN
			m_State_Axis2:=1;
		ELSE
			m_State_Axis2:=-100;
		END_IF
	1:
		//检查电机是否已经上电，如无，则上电
		IF 	NOT MC_Power_Axis2.Status THEN
			MC_Power_Axis2.Enable:=TRUE;
		ELSE
			m_State_Axis2:=2;
		END_IF
	2:
		//定位运行
		MC_MoveAbsolute_Axis2.Position:=targetPositionAxis2;
		MC_MoveAbsolute_Axis2.Velocity:=targetVelocityAxis2;
		IF btn_Move_Axis2 THEN
			MC_MoveAbsolute_Axis2.Execute:=TRUE;
			m_State_Axis2:=3;
		END_IF
	3:
		//是否运动到位
		IF MC_MoveAbsolute_Axis2.Done THEN
			m_State_Axis2:=88;
		END_IF
	88:
		btn_Move_Axis2:=FALSE;
		MC_MoveAbsolute_Axis2.Execute:=FALSE;
		m_State_Axis2:=0;		
	-100:
		btn_Move_Axis2:=FALSE;
		MC_MoveAbsolute_Axis2.Execute:=FALSE;
		Error:=TRUE;
		ErrorId:=1002;
		ErrorDescription:='E_STOP AND NOT Axis2_error';
		
END_CASE
//
//JOG+
//
CASE j_State_Axis2 OF 
	0:
		//检查是否有错误等
		IF  E_STOP  AND NOT Axis2_error THEN
			j_State_Axis2:=1;
		ELSE
			j_State_Axis2:=-100;
		END_IF
	1:
		//检查电机是否已经上电，如无，则上电
		IF 	NOT MC_Power_Axis2.Status THEN
			MC_Power_Axis2.Enable:=TRUE;
		ELSE
			j_State_Axis2:=2;
		END_IF
	2:
		//JOG运行
		MC_JOG_Axis2.Position:=increaseJogPositionAxis2;
		MC_JOG_Axis2.Velocity:=targetVelocityAxis2;
		IF btn_JogForward_Axis2 AND NOT btn_JogBackward_Axis2 THEN
			MC_JOG_Axis2.JogForward:=TRUE;
			j_State_Axis2:=3;
		END_IF
		IF btn_JogBackward_Axis2 AND NOT btn_JogForward_Axis2 THEN
			MC_JOG_Axis2.JogBackwards:=TRUE;
			j_State_Axis2:=3;
		END_IF
	3:
		//是否运动到位
		IF btn_JogForward_Axis2 THEN
			btn_JogForward_Axis2:=FALSE;
		END_IF 
		IF btn_JogBackward_Axis2 THEN
			btn_JogBackward_Axis2:=FALSE;
		END_IF
		IF MC_JOG_Axis2.Done THEN
			j_State_Axis2:=88;
		END_IF
	88:
		MC_JOG_Axis2.JogForward:=FALSE;
		MC_JOG_Axis2.JogBackwards:=FALSE;
		btn_JogForward_Axis2:=FALSE;
		btn_JogBackward_Axis2:=FALSE;
		j_State_Axis2:=0;	
		
	-100:
		MC_JOG_Axis2.JogForward:=FALSE;
		MC_JOG_Axis2.JogBackwards:=FALSE;
		btn_JogForward_Axis2:=FALSE;
		btn_JogBackward_Axis2:=FALSE;
		Error:=TRUE;
		ErrorId:=1002;
		ErrorDescription:='E_STOP AND NOT Axis2_error';	
END_CASE
//
//STOP
//
CASE s_State_Axis2 OF 
	0:
		//检查是否有错误等
		IF  E_STOP  AND NOT Axis2_error THEN
			s_State_Axis2:=1;
		ELSE
			s_State_Axis2:=-100;
		END_IF
	1:
		//检查电机是否已经上电，如无，则上电
		IF 	NOT MC_Power_Axis2.Status THEN
			MC_Power_Axis2.Enable:=TRUE;
		ELSE
			s_State_Axis2:=2;
		END_IF
	2:
		//STOP
		IF btn_Stop_Axis2 THEN
			MC_Stop_Axis2.Execute:=TRUE;
			s_State_Axis2:=3;
		END_IF
	3:
		//是否运动到位
		IF MC_Stop_Axis2.Done THEN
			s_State_Axis2:=88;
		END_IF
	88:
		btn_Stop_Axis2:=FALSE;
		MC_Stop_Axis2.Execute:=FALSE;
		s_State_Axis2:=0;	
		//reset status
		btn_Move_Axis2:=FALSE;
		MC_MoveAbsolute_Axis2.Execute:=FALSE;
		btn_JogForward_Axis2:=FALSE;
		btn_JogBackward_Axis2:=FALSE;
		MC_JOG_Axis2.JogForward:=FALSE;
		MC_JOG_Axis2.JogBackwards:=FALSE;
		m_State_Axis2:=0;
		j_State_Axis2:=0;
	-100:
		btn_Stop_Axis2:=FALSE;
		MC_Stop_Axis2.Execute:=FALSE;
		Error:=TRUE;
		ErrorId:=1002;
		ErrorDescription:='E_STOP AND NOT Axis2_error';
		//reset status
		btn_Move_Axis2:=FALSE;
		MC_MoveAbsolute_Axis2.Execute:=FALSE;
		btn_JogForward_Axis2:=FALSE;
		btn_JogBackward_Axis2:=FALSE;
		MC_JOG_Axis2.JogForward:=FALSE;
		MC_JOG_Axis2.JogBackwards:=FALSE;
		m_State_Axis2:=0;
		j_State_Axis2:=0;
END_CASE
//
//Reset
//
CASE r_State_Axis2 OF 
	0:
		IF btn_Reset_Axis2 THEN
			MC_Reset_Axis2.Execute:=TRUE;
			r_State_Axis2:=1;
		END_IF
	1:
		//是否运动到位
		IF MC_Reset_Axis2.Done THEN
			r_State_Axis2:=88;
		END_IF
	88:
		r_State_Axis2:=0;
		MC_Reset_Axis2.Execute:=FALSE;	
		btn_Reset_Axis2:=FALSE;
		//reset status
		btn_Move_Axis2:=FALSE;
		MC_MoveAbsolute_Axis2.Execute:=FALSE;
		btn_JogForward_Axis2:=FALSE;
		btn_JogBackward_Axis2:=FALSE;
		MC_JOG_Axis2.JogForward:=FALSE;
		MC_JOG_Axis2.JogBackwards:=FALSE;
		m_State_Axis2:=0;
		s_State_Axis2:=0;
		j_State_Axis2:=0;
END_CASE
//
//setposotion
//
SetPosition_delay_Axis2.PT:=T#0.1S;
SetPosition_delay_Axis2();
IF btn_SetPosition_Axis2 THEN
	CASE sp_State_Axis2 OF 
		0:
			IF NOT Axis2_moving THEN
				sp_State_Axis2:=1;
			END_IF
		1:
			MC_SetPosition_Axis2.Position:=PositionSetValue_Axis2;
			MC_SetPosition_Axis2.Execute:=TRUE;
			SetPosition_delay_Axis2.IN:=TRUE;
			sp_State_Axis2:=2;
		2:
			IF MC_SetPosition_Axis2.Done THEN
				sp_State_Axis2:=88;
			END_IF
			IF SetPosition_delay_Axis2.Q THEN//延时结束时，还没有设置位置成功
				sp_State_Axis2:=-100;
			END_IF
		88:
			PositionSetDone_Axis2:=TRUE;
			MC_SetPosition_Axis2.Execute:=FALSE;
			SetPosition_delay_Axis2.IN:=FALSE;
			sp_State_Axis2:=0;
			btn_SetPosition_Axis2:=FALSE;
		-100:
			PositionSetDone_Axis2:=FALSE;
			MC_SetPosition_Axis2.Execute:=FALSE;
			SetPosition_delay_Axis2.IN:=FALSE;
			btn_SetPosition_Axis2:=FALSE;
	END_CASE
END_IF
//
//屏幕按钮**互锁变量,FALSE时，该按钮灰色不能触发
//
//J1->JOG+
IF  foreward_limit_axis1 AND E_STOP  AND Local_led AND NOT  Axis2_error  AND NOT  Axis2_moving AND
	NOT btn_Move_Axis2 AND NOT  btn_JogBackward_Axis2  THEN
	Axis2_J1     := TRUE;
ELSE
	Axis2_J1     := FALSE;
END_IF;
//J2>JOG-
IF  backward_limit_axis1  AND E_STOP   AND Local_led AND NOT  Axis2_error  AND NOT  Axis2_moving AND 
	 NOT  btn_Move_Axis2 AND NOT btn_JogForward_Axis2 THEN
	Axis2_J2     := TRUE;
ELSE
	Axis2_J2     := FALSE;
END_IF;
//P->PositionMove
IF  E_STOP   AND Local_led AND NOT  Axis2_error  AND NOT  Axis2_moving AND 
	 NOT btn_JogForward_Axis2  AND NOT  btn_JogBackward_Axis2 THEN
	Axis2_P     := TRUE;
ELSE
	Axis2_P     := FALSE;
END_IF;
//SP->SetPosition
IF E_STOP  AND Local_led AND NOT  Axis2_error  AND NOT Axis2_moving  THEN
	Axis2_SP     := TRUE;
ELSE
	Axis2_SP     := FALSE;
END_IF;
//S->Stop
IF E_STOP  AND Local_led AND NOT  Axis2_error THEN
	Axis2_S     := TRUE;
ELSE
	Axis2_S     := FALSE;
END_IF;
//
//
//
//急停
E_STOP_ftring(CLK:=E_STOP , Q=> );
E_STOP_rem_ftring(CLK:=E_STOP_rem , Q=> );
IF E_STOP_ftring.Q OR E_STOP_rem_ftring.Q THEN     
	E_STOP_led:= TRUE;	
	MC_Power_Axis2.Enable:=FALSE;//电机2断电
	btn_Stop_Axis2:=TRUE;//STOP axis1
	A_MCAxis2();
	Error:=TRUE;
	ErrorId:=101;
	ErrorDescription:='E_STOP';
END_IF;

ACTION A_MCAxis2:
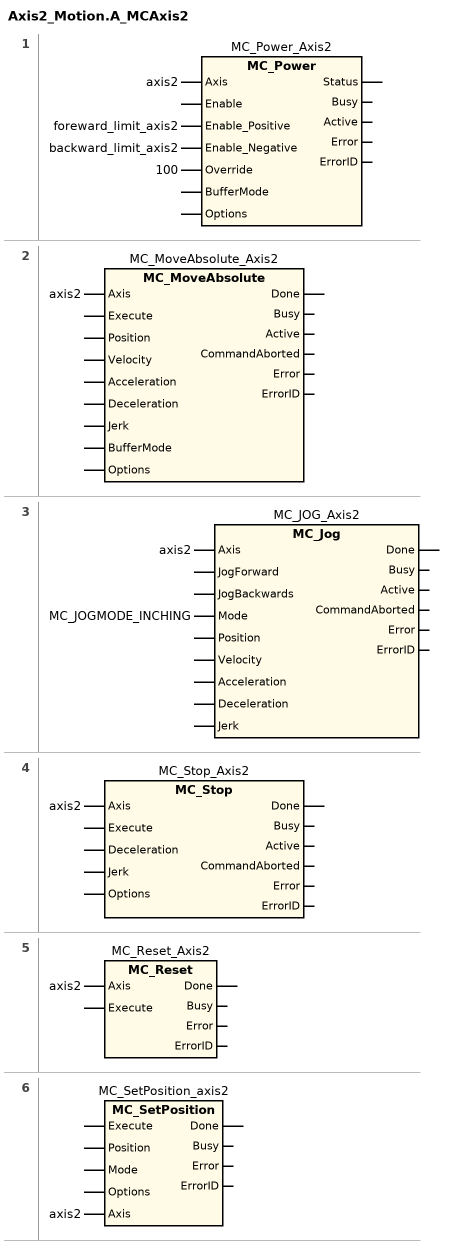
// NETWORK 1
MC_Power_Axis2(
    Axis := axis2,
    Enable_Positive := foreward_limit_axis2,
    Enable_Negative := backward_limit_axis2,
    Override := 100); // MC_Power

// NETWORK 2
MC_MoveAbsolute_Axis2(Axis := axis2); // MC_MoveAbsolute

// NETWORK 3
MC_JOG_Axis2(Axis := axis2, Mode := MC_JOGMODE_INCHING); // MC_Jog

// NETWORK 4
MC_Stop_Axis2(Axis := axis2); // MC_Stop

// NETWORK 5
MC_Reset_Axis2(Axis := axis2); // MC_Reset

// NETWORK 6
MC_SetPosition_axis2(Axis := axis2); // MC_SetPosition
END_ACTION

END_PROGRAM
